VAR_GLOBAL CONSTANT
	


END_VAR

(* stored: Version 1.1.0.1, ProductVersion 3.1.4024.9
   GVL GVL_CONSTANT: Id {7419296d-3549-414c-8cb8-622088338c3b} *)
